FUNCTION_BLOCK T_MoveCylinderToPosition IMPLEMENTS I_CylinderMover, ITaskStatus
VAR
	_actuatorToSet : REFERENCE TO BOOL;
	_actuatorToClear : REFERENCE TO BOOL;
	_atPositionSensor : REFERENCE TO BOOL;	
	_move : BOOL;
	moveTimeout : TON;
END_VAR

_actuatorToSet S= _move;
_actuatorToClear R= _move;
_move R= _atPositionSensor; 
moveTimeout( IN := _move );

METHOD Abort
_move := FALSE;
END_METHOD

PROPERTY Busy : BOOL
GET
Busy := _move;
END_GET
END_PROPERTY

PROPERTY Done : BOOL
GET
Done := _atPositionSensor;
END_GET
END_PROPERTY

PROPERTY Error : BOOL
GET
Error := moveTimeout.Q;
END_GET
END_PROPERTY

METHOD FB_init : BOOL
VAR_INPUT
	bInitRetains : BOOL; // if TRUE, the retain variables are initialized (warm start / cold start)
	bInCopyCode : BOOL;  // if TRUE, the instance afterwards gets moved into the copy code (online change)
	actuatorToSet : REFERENCE TO BOOL;   
	actuatorToClear : REFERENCE TO BOOL; 
	atPositionSensor : REFERENCE TO BOOL;
	moveTimeoutErr : TIME;
END_VAR
moveTimeout.PT := moveTimeoutErr;
_actuatorToSet REF= actuatorToSet;
_actuatorToClear REF=  actuatorToClear;
_atPositionSensor REF= atPositionSensor;
END_METHOD

METHOD PUBLIC MoveToTarget : BOOL
IF Busy THEN
	RETURN;
END_IF

MoveToTarget := _move := TRUE;
END_METHOD

END_FUNCTION_BLOCK

(* stored: Version 1.1.0.1, ProductVersion 3.1.4024.4
   POU T_MoveCylinderToPosition: Id {02039554-bb19-4a40-8b78-b2344b5ef1db}, SpecialFunc None
   Method Abort: Id {5c1f8582-8e40-45d4-9c60-d868d00b7b54}
   Property Busy: Id {a8683767-ee4e-4b5f-bead-c7f729b17dd3}
   Get Get: Id {ee494e21-dd22-4d40-afe9-71bc4bd7dbdb}
   Property Done: Id {15b19d75-8ca1-458c-811e-9dbc7b43ed89}
   Get Get: Id {cf1b6bf3-69e6-42e3-8a4d-aa62a891cf38}
   Property Error: Id {148dc56c-3bdf-4996-80a1-e79cb0f0663b}
   Get Get: Id {f8df5910-601c-4e00-8347-72e7109b1272}
   Method FB_init: Id {9927bf8c-2c75-48f0-bf3b-1663a42da55e}
   Method MoveToTarget: Id {71ad3fcd-a2a2-4893-9198-a4a13f4ffbc2} *)
